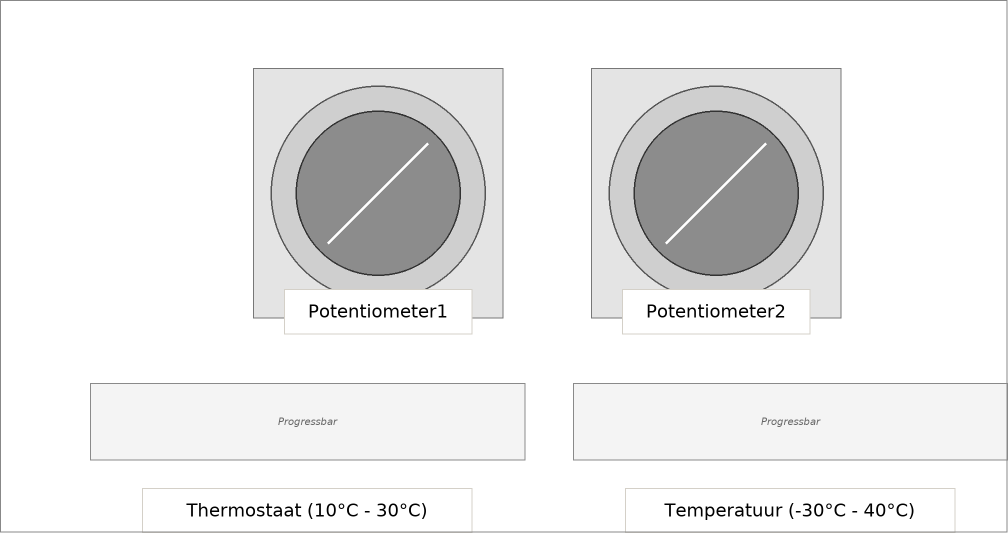
VISUALIZATION Visualization_Thermostaatregeling  // 1008x533
    Potentiometer360 (253,68 250x250), variable: prg_Thermostaatregeling.Potentiometer1, style: Potentiometer-Potentiometer360-Gray, scale format: %.1f, scale 10..30
        p2431819421: Outside
    Potentiometer360 (591,68 250x250), variable: prg_Thermostaatregeling.Potentiometer2, style: Potentiometer-Potentiometer360-Gray, scale format: %.1f, scale -30..40
        p2431819421: Outside
    Textfield (284,289 188x45), "Potentiometer1"
    Textfield (622,289 188x45), "Potentiometer2"
    Progressbar (573,383 435x77), variable: prg_Thermostaatregeling.Temperatuur
    Textfield (625,488 330x45), "Temperatuur (-30°C - 40°C)"
    Progressbar (90,383 435x77), variable: prg_Thermostaatregeling.Temperatuur
    Textfield (142,488 330x45), "Thermostaat (10°C - 30°C)"
END_VISUALIZATION

(* stored: Version 1.1.0.1, ProductVersion 3.1.4024.15
   Visu Visualization_Thermostaatregeling: Id {13216c18-555a-4df1-85a6-a8597b89ee8b} *)
